FUNCTION_BLOCK FB_System_Fenster
VAR_INPUT
	Freigabe_auto			: BOOL;
	Quittierung				: BOOL;
	Betrieb_Anford_auto			: BOOL;
	Parameter_init			: ST_System_Fenster_Parameter;
END_VAR
VAR_OUTPUT
	{attribute 'OPC.UA.DA' := '1'}Parameter				: ST_System_Fenster_Parameter;		
	{attribute 'OPC.UA.DA' := '1'}Steuerung				: ST_System_Fenster_Steuerung;		
	{attribute 'OPC.UA.DA' := '1'}Stellwert				: ST_System_Fenster_Stellwert;		
	{attribute 'OPC.UA.DA' := '1'}Zustand					: ST_System_Fenster_Zustand;	
END_VAR
VAR
	IN_Servomotor_Fenster_O_W_auf			AT %I*: BOOL;
	IN_Oberlichter_Halle_Stellung			AT %I*: BOOL;
	IN_Oberlichter_Treppenhaus_Stellung		AT %I*: BOOL;

	Fenster_Halle_OST		: FB_Fenster;
	Fenster_Halle_WEST		: FB_Fenster;
	Lesedaten				: FB_Fenster_Input;
	test: BOOL;
	test1: BOOL;
	test2: BOOL;
	Regelung: FB_System_Fenster_Regelung;
	Logik: FB_System_Fenster_Logik;
END_VAR

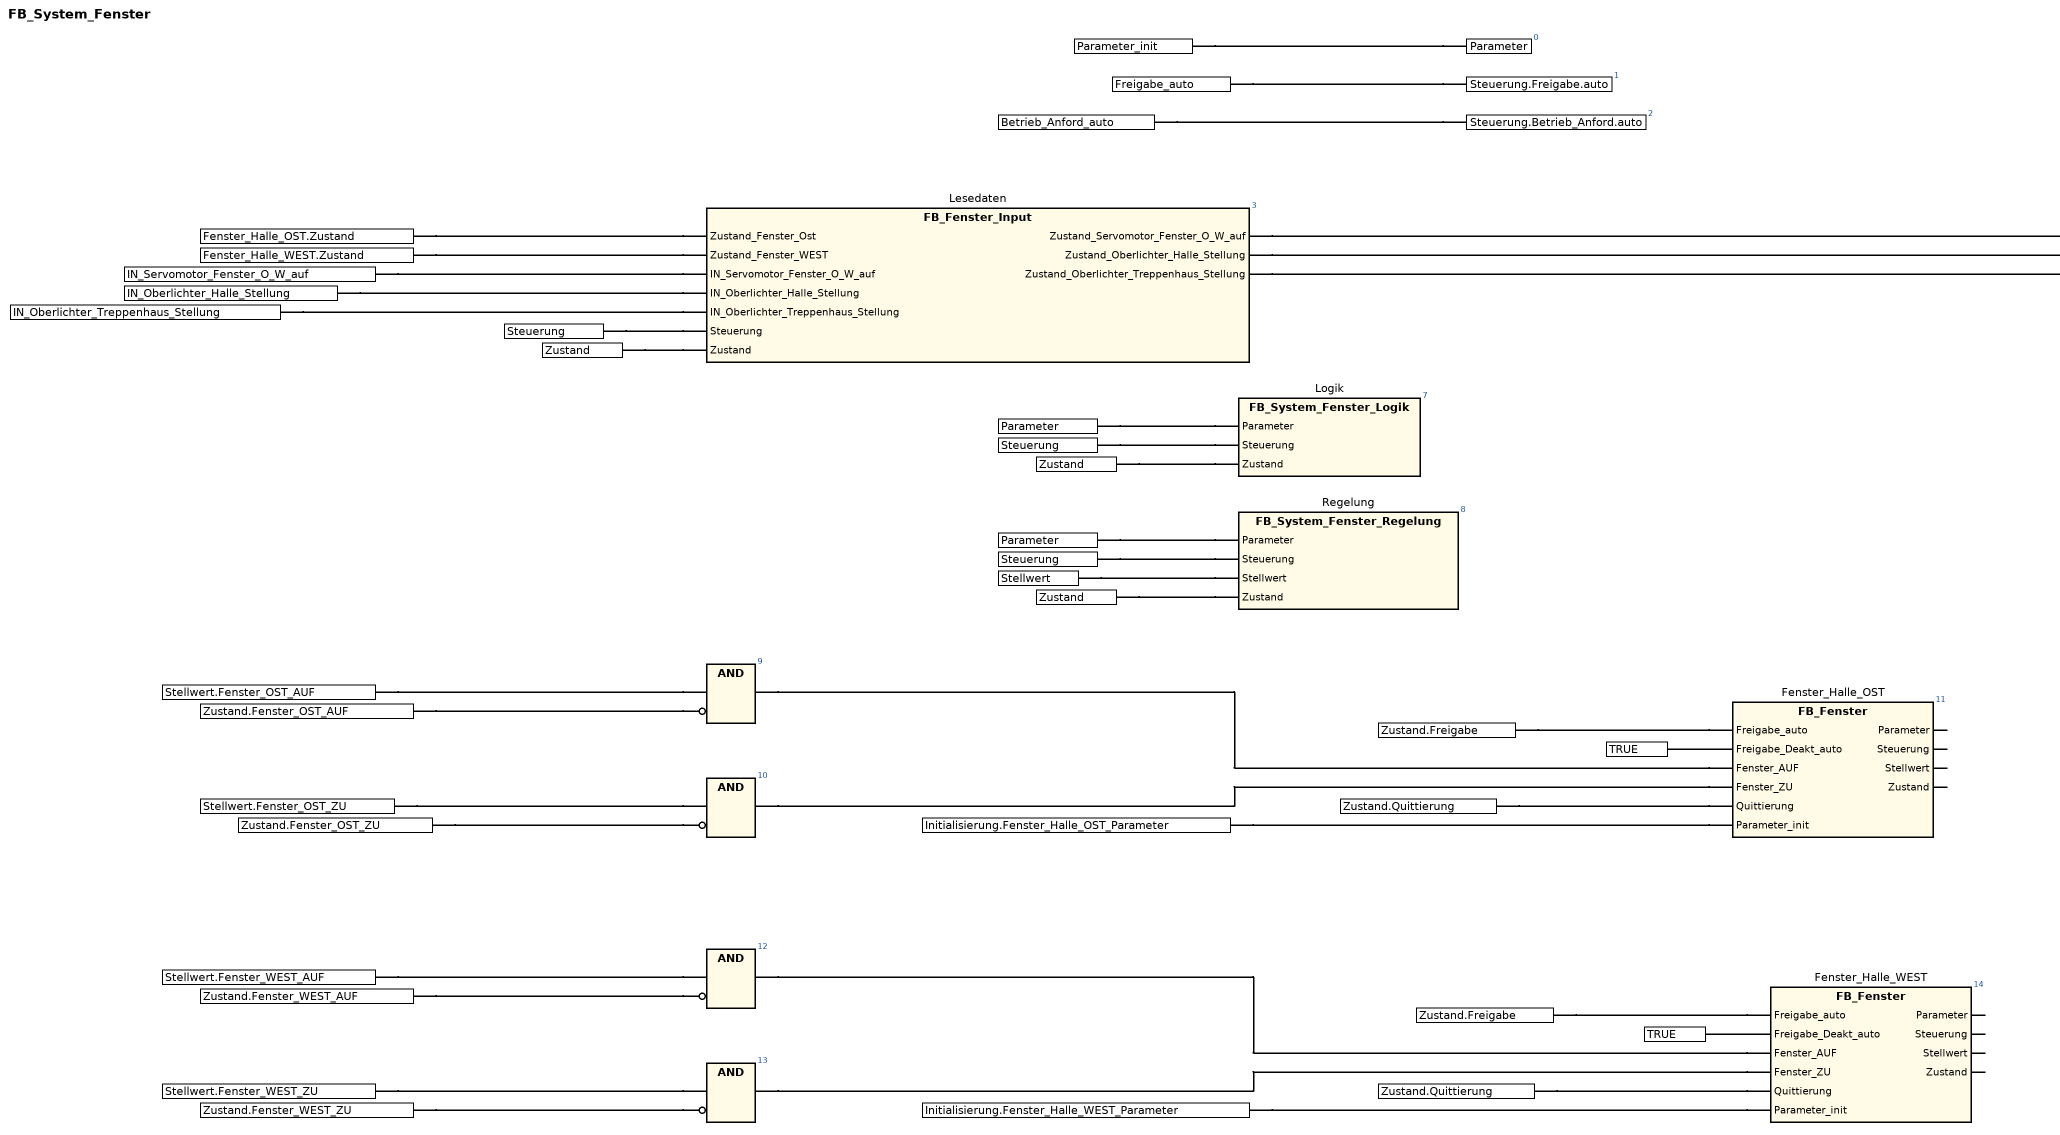
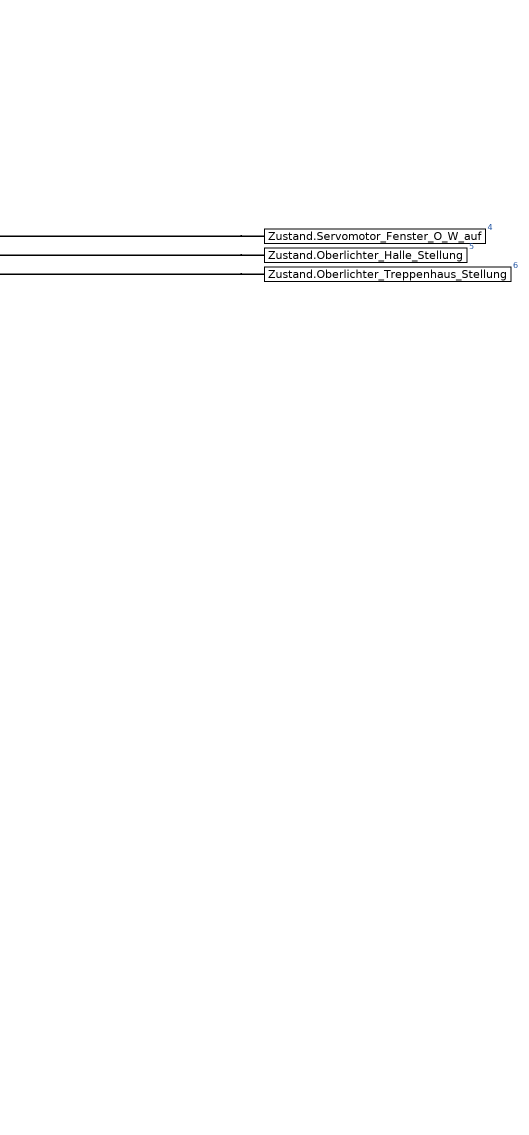
Parameter := Parameter_init;
Steuerung.Freigabe.auto := Freigabe_auto;
Steuerung.Betrieb_Anford.auto := Betrieb_Anford_auto;
Lesedaten(
    Zustand_Fenster_Ost := Fenster_Halle_OST.Zustand,
    Zustand_Fenster_WEST := Fenster_Halle_WEST.Zustand,
    IN_Servomotor_Fenster_O_W_auf := IN_Servomotor_Fenster_O_W_auf,
    IN_Oberlichter_Halle_Stellung := IN_Oberlichter_Halle_Stellung,
    IN_Oberlichter_Treppenhaus_Stellung := IN_Oberlichter_Treppenhaus_Stellung,
    Steuerung := Steuerung,
    Zustand := Zustand); // FB_Fenster_Input
Zustand.Servomotor_Fenster_O_W_auf := Lesedaten.Zustand_Servomotor_Fenster_O_W_auf;
Zustand.Oberlichter_Halle_Stellung := Lesedaten.Zustand_Oberlichter_Halle_Stellung;
Zustand.Oberlichter_Treppenhaus_Stellung := Lesedaten.Zustand_Oberlichter_Treppenhaus_Stellung;
Logik(Parameter := Parameter, Steuerung := Steuerung, Zustand := Zustand); // FB_System_Fenster_Logik
Regelung(Parameter := Parameter, Steuerung := Steuerung, Stellwert := Stellwert, Zustand := Zustand); // FB_System_Fenster_Regelung
Fenster_Halle_OST(
    Freigabe_auto := Zustand.Freigabe,
    Freigabe_Deakt_auto := TRUE,
    Fenster_AUF := Stellwert.Fenster_OST_AUF AND NOT Zustand.Fenster_OST_AUF,
    Fenster_ZU := Stellwert.Fenster_OST_ZU AND NOT Zustand.Fenster_OST_ZU,
    Quittierung := Zustand.Quittierung,
    Parameter_init := Initialisierung.Fenster_Halle_OST_Parameter); // FB_Fenster
Fenster_Halle_WEST(
    Freigabe_auto := Zustand.Freigabe,
    Freigabe_Deakt_auto := TRUE,
    Fenster_AUF := Stellwert.Fenster_WEST_AUF AND NOT Zustand.Fenster_WEST_AUF,
    Fenster_ZU := Stellwert.Fenster_WEST_ZU AND NOT Zustand.Fenster_WEST_ZU,
    Quittierung := Zustand.Quittierung,
    Parameter_init := Initialisierung.Fenster_Halle_WEST_Parameter); // FB_Fenster

END_FUNCTION_BLOCK

(* stored: Version 1.1.0.1, ProductVersion 3.1.4024.9
   POU FB_System_Fenster: Id {cf80e2b7-0352-4ad5-8410-3d4bcb744ee7}, SpecialFunc None *)
